TYPE (* A Directly Derived Data Type *)
  (* Standard: 61499-2 *)
  (* Version 0.0, 2003-12-06, JHC, Rockwell Automation *)
  (* Compiler header: package fb.rt.template; *)
  (* ASN.1 tag PRIVATE 7 *)
  Direct : REAL := 5.1;
END_TYPE
